FUNCTION_BLOCK CAT_Conveyor_HMI (* Service Interface Function Block Type *)
  (* Standard: 61499-2 *)
  (* Version 0.0, 16/08/2021, prana, nxtControl GmBH, template *)
  PACKAGE Main;
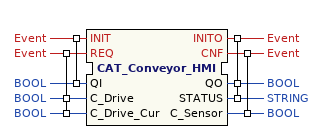
  EVENT_INPUT
    INIT WITH QI;
    REQ WITH C_Drive, C_Drive_Cur;
  END_EVENT
  EVENT_OUTPUT
    INITO WITH QO, STATUS;
    CNF WITH C_Sensor;
  END_EVENT
  VAR_INPUT
    QI : BOOL;
    C_Drive : BOOL;
    C_Drive_Cur : BOOL;
  END_VAR
  VAR_OUTPUT
    QO : BOOL; (* Event Output Qualifier *)
    STATUS : STRING; (* Service Status *)
    C_Sensor : BOOL;
  END_VAR
  SERVICE /
    SEQUENCE 
    END_SEQUENCE
  END_SERVICE
END_FUNCTION_BLOCK
